// TIA Portal V19 export
FUNCTION "A0304_Manager_CALL" : Void   // FC192, LAD
TITLE = Manager AREA 304
// stored: SetENOAutomatically false
BEGIN

REGION Network 1 (SCL): << TRASFERIMENTO stati CIn del blocco >>
   // // TRASFERIMENTO CIn Navetta
   "A0304_Manager".CIn.Navetta := "A0304_Navetta".COut;

   //TRASFERIMENTO Cin Sollevamento
   "A0304_Manager".CIn.Sollevamento.ReadyToDrop := "A0303_Manager".Sts.Sollevatore.InPosDeposito OR "A0303_Manager".Sts.Sollevatore.InPosPreDeposito ; //(("BTrk".A0303.Stacker.Layers_Qty >= "BTrk".A0303.Stacker.Layers_Target) OR "BTrk".A0303.Stacker.Completato ) AND "A0303_Manager".Sts.Sollevatore.InPosDeposito ;

   "A0304_Manager".CIn.Antiribaltamento.Rest :="A0303_Manager".Sts.SostegnoTesta.Ax.InRestPos AND "A0303_Manager".Sts.SostegnoCoda.Ax.InRestPos AND "A0303_Sostegno_Testa".COut.Paletto.RestPosition AND "A0303_Sostegno_Coda".COut.Paletto.RestPosition;
   "A0304_Manager".CIn.Antiribaltamento.PalettoPos0 := "A0303_Sostegno_Testa".COut.Paletto.RestPosition AND "A0303_Sostegno_Coda".COut.Paletto.RestPosition;


   // Mng 03
   "A0304_Manager".CIn.Manager03.IsWaiting_NoPiecesBefore := "A0303_Manager".Warning.IsWaiting_NoPiecesBefore;

   // Production Mng
   "A0304_Manager".CIn.ProdManager := "Areas_ITF".Prod.A03_A04;
END_REGION

REGION Network 2: DataIn
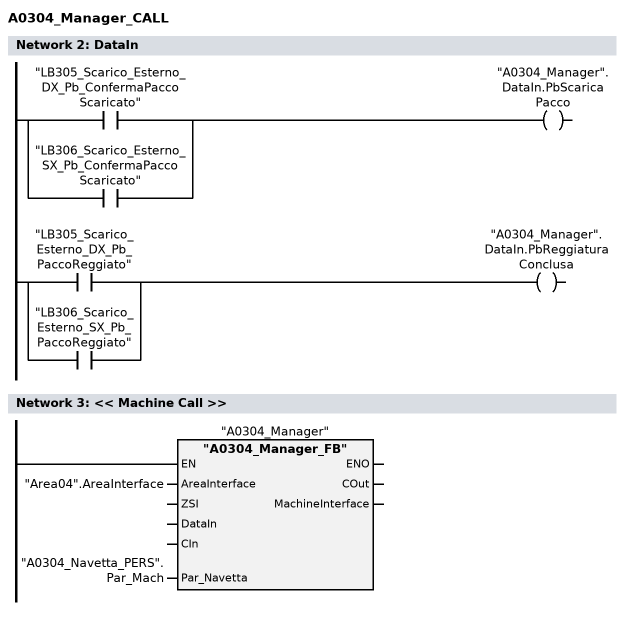
   RUNG wire#powerrail
      Contact( "LB305_Scarico_Esterno_DX_Pb_ConfermaPaccoScaricato" )
      wire#w1
      Coil( "A0304_Manager".DataIn.PbScaricaPacco )
   END_RUNG
   RUNG wire#powerrail
      Contact( "LB306_Scarico_Esterno_SX_Pb_ConfermaPaccoScaricato" )
   END_RUNG wire#w1
   RUNG wire#powerrail
      Contact( "LB305_Scarico_Esterno_DX_Pb_PaccoReggiato" )
      wire#w2
      Coil( "A0304_Manager".DataIn.PbReggiaturaConclusa )
   END_RUNG
   RUNG wire#powerrail
      Contact( "LB306_Scarico_Esterno_SX_Pb_PaccoReggiato" )
   END_RUNG wire#w2
   // the same network as SCL:
   "A0304_Manager".DataIn.PbScaricaPacco := "LB305_Scarico_Esterno_DX_Pb_ConfermaPaccoScaricato" OR "LB306_Scarico_Esterno_SX_Pb_ConfermaPaccoScaricato";
   "A0304_Manager".DataIn.PbReggiaturaConclusa := "LB305_Scarico_Esterno_DX_Pb_PaccoReggiato" OR "LB306_Scarico_Esterno_SX_Pb_PaccoReggiato";
END_REGION

REGION Network 3: << Machine Call >>
   RUNG wire#powerrail
      "A0304_Manager"(AreaInterface := "Area04".AreaInterface, ZSI :=, DataIn :=, CIn :=, Par_Navetta := "A0304_Navetta_PERS".Par_Mach, COut =>, MachineInterface =>)
   END_RUNG
   // the same network as SCL:
   "A0304_Manager"(AreaInterface := "Area04".AreaInterface, Par_Navetta := "A0304_Navetta_PERS".Par_Mach);   // "A0304_Manager_FB"
END_REGION

REGION Network 4 (SCL): << OP CND >>
   //Vai a Prelievo
   "A0304_Manager".OP_CND.VaiAPrelievo[0].Visible := TRUE;
   "A0304_Manager".OP_CND.VaiAPrelievo[0].Condition := "BTrk".A0304.Empty;
   "A0304_Manager".OP_CND.VaiAPrelievo[0].Description :='Assenza Trk nu navetta';

   "A0304_Manager".OP_CND.VaiAPrelievo[1].Visible := TRUE;
   "A0304_Manager".OP_CND.VaiAPrelievo[1].Condition := "A0304_Manager".Sts.InPosPrePrelievo;
   "A0304_Manager".OP_CND.VaiAPrelievo[1].Description := 'Non in posizione di prelievo';
END_REGION
END_FUNCTION
